TYPE ST_AX5000Diag :
STRUCT
(* NC-Status *)
	nNCAxisID							: UDINT;
	bOperational						: BOOL;
	bC1DError							: BOOL;
	bWcStateError						: BOOL;
	bAxisError							: BOOL;
	iAxisErrorCode						: UDINT;

(* Drive Diag *)
	strDriveType						: STRING(19);
	strMotorType						: STRING(31);
	wDriveStatus						: WORD;
	wClass1Diag							: WORD;
	stClass1Diag						: ST_AX5000_C1D;
	stDriveStatus						: ST_AX5000DriveStatus;
	stEcSlaveStateBits					: ST_EcSlaveStateBits;
	stEcSlaveState						: ST_EcSlaveState;
	bPreopToSafeOpError					: BOOL;
	bSafeOpToOpError					: BOOL;
	stCPxInvParamList					: ST_SoE_CPxInvParamList;
	iDiagNumber							: UDINT;
	stDiagNumberList					: ST_SoE_DiagNumList;
	strDiagMessage						: STRING;
END_STRUCT
END_TYPE

(* stored: Version 1.1.0.1, ProductVersion 3.1.4026.13, FileIdentifier 67b9bef29b8b5b833f1e44246a041aa2ee723353, FileSignature 538025c4ccae232e89c003d27f6abafdafb21d8063ef331b9f512e8a4d22dd0b18e772ec630c48724cde3ad85a1c2f8fe82319d793c73c38dabae5dd4439dcf3ee0299cbffbd6a5e218d3c715acd91d8eea0b4441cab941e78ef0459eb17304a83a47b29e0c2b9c59335d48133766f357f2b8a7208dd07139a4a1e79f952548eb7b63da2be0fedfca89217a1c0b7d4d3732404441ddd71b38ed8710310cbcb7a431c32d23a2c7686957a379ee8084a45c9211dd9a2a13d140804516f288422b09ed198b84f8b8d761189c29163e01822ec0b1da1bc6aa3783c8d1c51947c0431ba37dbf1e5e385191744fc7d88845bc9b21613308ebff5497841995c68e325c4
   DUT ST_AX5000Diag: Id {652333d8-1c07-47ed-9bf7-2897e05e7d36} *)
